PROGRAM MAIN
VAR
END_VAR

END_PROGRAM

(* stored: Version 1.1.0.1
   POU MAIN: Id {ee31915d-83fa-4a0b-bf8e-4c43484669b5} *)
